FUNCTION_BLOCK FB_Pump
VAR_INPUT
END_VAR
VAR_OUTPUT
END_VAR
VAR
	rStartSpeed		: UINT;		//Startdrehzahl 0..100%
	rRatedSpeed		: UINT;		//Nenndrehzahl 0..100%
	tStartDelay		: TIME;		//Delay Startdrehzahl -> Nenndrehzahl
	timer			: TON;		
	bIsOn			: BOOL;
	//Ausgänge für Geräteverknüpfung
	bDigiOut	 	AT %Q* : BOOL;		//Standardpumpe EIN/AUS
	nPWMValue 		AT %Q* : UINT;	//PWM für Drehzahl
END_VAR

METHOD M_On : BOOL
VAR_INPUT
END_VAR
bDigiOut := TRUE;
IF tStartDelay > T#0S AND NOT bIsOn THEN
	nPWMValue := REAL_TO_UINT(32767.0 / 100 * rStartSpeed);
	timer(IN:=TRUE,PT:= tStartDelay);
	IF timer.Q THEN
		timer(IN:=FALSE);
		nPWMValue := REAL_TO_UINT(32767.0 / 100 * rRatedSpeed);
		M_On := TRUE;	
	END_IF
ELSE
	nPWMValue := REAL_TO_UINT(32767.0 / 100 * rRatedSpeed);
	M_On := TRUE;
	bIsOn := TRUE;
END_IF
END_METHOD

PROPERTY P_bIsOn : BOOL
GET
P_bIsOn := bDigiOut;
END_GET
END_PROPERTY

PROPERTY P_nStartSpeed : USINT
SET
IF P_nStartSpeed <= 100 THEN
	rStartSpeed := P_nStartSpeed; 
ELSE
	rStartSpeed := 100;
END_IF
END_SET
END_PROPERTY

PROPERTY P_nRatedSpeed : USINT
SET
IF P_nRatedSpeed <= 100 THEN
	rRatedSpeed := P_nRatedSpeed; 
ELSE
	rRatedSpeed := 100;
END_IF
END_SET
END_PROPERTY

PROPERTY P_nDelay : UINT
SET
tStartDelay := UINT_TO_TIME(P_nDelay);
END_SET
END_PROPERTY

METHOD M_Off
VAR_INPUT
END_VAR
bDigiOut := FALSE;
nPWMValue := 0;
timer(IN:=FALSE);
bIsOn := FALSE;
END_METHOD

END_FUNCTION_BLOCK

(* stored: Version 1.1.0.1, ProductVersion 3.1.4020.6
   POU FB_Pump: Id {6a5a5d39-6556-4708-b72c-bd2317235676}, SpecialFunc None
   Method M_On: Id {11b885ac-9d26-47b2-b01f-bba258325c54}
   Property P_bIsOn: Id {18eeca7b-b384-433b-952c-d33672c388e9}
   Get Get: Id {f5a00200-f941-4414-a47d-b93dbecdeb0a}
   Property P_nStartSpeed: Id {7c1a9499-a688-45ba-92d8-d0e76ae6731e}
   Set Set: Id {294075a5-b959-440d-8cf6-141d6cf9750d}
   Property P_nRatedSpeed: Id {8556d0b7-6163-4ace-8e41-8cf29a249619}
   Set Set: Id {f6cd64ed-d870-4d99-adcd-2727a476a648}
   Property P_nDelay: Id {d182ac0d-3f99-4ab8-9423-8a9206fd19af}
   Set Set: Id {6f3554b7-9c8f-4430-bbdf-06142a308e2c}
   Method M_Off: Id {f2ede433-4556-404c-a985-dd6f1d73cd7c} *)
